GLOBALCONSTANTS IG3_NAME_Functions (* Industry Group 3 specific function defines *)
  (* Standard: 61499-1 *)
  (* Version 1.0, 2026-06-29, Franz Höpfinger, Demmler Andreas Fahrzeugbau *)
  PACKAGE isobus::pgn::const;
  VAR_GLOBAL CONSTANT
    F_SUPPLEMENTAL_ENGINE_CONTROL_SENSING : BYTE := 128; (* Sys: Non-specific system, Func: Supplemental Engine Control Sensing *)
    F_LASER_RECEIVER : BYTE := 129; (* Sys: Non-specific system, Func: Laser Receiver *)
    F_LAND_LEVELING_SYSTEM_OPERATOR_INTERFACE : BYTE := 130; (* Sys: Non-specific system, Func: Land Leveling System Operator Interface - A component that allows *)
    F_LAND_LEVELING_ELECTRIC_MAST : BYTE := 131; (* Sys: Non-specific system, Func: Land Leveling Electric Mast *)
    F_SINGLE_LAND_LEVELING_SYSTEM_SUPERVISOR : BYTE := 132; (* Sys: Non-specific system, Func: Single Land Leveling System Supervisor *)
    F_LAND_LEVELING_SYSTEM_DISPLAY : BYTE := 133; (* Sys: Non-specific system, Func: Land Leveling System Display *)
    F_LASER_TRACER : BYTE := 134; (* Sys: Non-specific system, Func: Laser Tracer *)
    F_LOADER_CONTROL : BYTE := 135; (* Sys: Non-specific system, Func: Loader Control *)
    F_SLOPE_SENSOR : BYTE := 136; (* Sys: Non-specific system, Func: Slope Sensor - Measures the slope along a axis. *)
    F_LIFTARM_CONTROL : BYTE := 137; (* Sys: Non-specific system, Func: Liftarm Control - Controller whose primary purpose is to control *)
    F_SUPPLEMENTAL_SENSOR_PROCESSING_UNITS : BYTE := 138; (* Sys: Non-specific system, Func: Supplemental Sensor Processing Units - An ECU functioning as an *)
    F_HYDRAULIC_SYSTEM_PLANNER : BYTE := 139; (* Sys: Non-specific system, Func: Hydraulic System Planner - Coordinates the functions of a number *)
    F_HYDRAULIC_VALVE_CONTROLLER : BYTE := 140; (* Sys: Non-specific system, Func: Hydraulic Valve Controller - The valve controller will typically *)
    F_JOYSTICK_CONTROL : BYTE := 141; (* Sys: Non-specific system, Func: Joystick Control - Joystick Control *)
    F_ROTATION_SENSOR : BYTE := 142; (* Sys: Non-specific system, Func: Rotation Sensor - A device that measures the rotational angle *)
    F_SONIC_SENSOR : BYTE := 143; (* Sys: Non-specific system, Func: Sonic Sensor - A device that measures distance via ultrasonic *)
    F_SURVEY_TOTAL_STATION_TARGET : BYTE := 144; (* Sys: Non-specific System, Func: Survey Total Station Target - A survey total station target shall *)
    F_HEADING_SENSOR : BYTE := 145; (* Sys: Non-specific System, Func: Heading Sensor - A device that measures vehicle azimuth. *)
    F_ALARM_DEVICE : BYTE := 146; (* Sys: Non-specific System, Func: Alarm device - Device that provides an audible and/or visual *)
    F_NOT_AVAILABLE : BYTE := 255; (* Sys: Non-specific system, Func: Not Available - This assignment can be used until an explicit *)
    F_SKID_STEER_LOADER_MAIN_CONTROLLER : BYTE := 128; (* Sys: Skid Steer Loader, Func: Main Controller *)
    F_SKID_STEER_LOADER_NOT_AVAILABLE : BYTE := 255; (* Sys: Skid Steer Loader, Func: Not Available - This assignment can be used until an explicit *)
    F_ARTICULATED_DUMP_TRUCK_NOT_AVAILABLE : BYTE := 255; (* Sys: Articulated Dump Truck, Func: Not Available - This assignment can be used until an explicit *)
    F_BACKHOE_NOT_AVAILABLE : BYTE := 255; (* Sys: Backhoe, Func: Not Available - This assignment can be used until an explicit function has *)
    F_CRAWLER_BLADE_CONTROLLER : BYTE := 128; (* Sys: Crawler, Func: Blade Controller - Controller for blade height. *)
    F_CRAWLER_NOT_AVAILABLE : BYTE := 255; (* Sys: Crawler, Func: Not Available - This assignment can be used until an explicit function has *)
    F_EXCAVATOR_SLOPE_SENSOR : BYTE := 128; (* Sys: Excavator, Func: Slope Sensor - Measures the slope along a axis. *)
    F_EXCAVATOR_NOT_AVAILABLE : BYTE := 255; (* Sys: Excavator, Func: Not Available - This assignment can be used until an explicit function has *)
    F_FORKLIFT_NOT_AVAILABLE : BYTE := 255; (* Sys: Forklift, Func: Not Available - This assignment can be used until an explicit function has *)
    F_FOUR_WHEEL_DRIVE_LOADER_NOT_AVAILABLE : BYTE := 255; (* Sys: Four Wheel Drive Loader, Func: Not Available - This assignment can be used until an explicit *)
    F_GRADER_HFWD_CONTROLLER : BYTE := 128; (* Sys: Grader, Func: HFWD Controller - Hydraulic front wheel drive controller *)
    F_GRADER_NOT_AVAILABLE : BYTE := 255; (* Sys: Grader, Func: Not Available - This assignment can be used until an explicit function has *)
    F_MILLING_MACHINE_NOT_AVAILABLE : BYTE := 255; (* Sys: Milling Machine, Func: Not Available - The milling machine is used for cutting (or chipping) *)
    F_RECYCLER_AND_SOIL_STABILIZER_NOT_AVAILABLE : BYTE := 255; (* Sys: Recycler and Soil Stabilizer, Func: Not Available - Cold recyclers are used to prepare the *)
    F_BINDING_AGENT_SPREADER_NOT_AVAILABLE : BYTE := 255; (* Sys: Binding Agent Spreader, Func: Not Available - Spreading large quantities of binding agents *)
    F_PAVER_NOT_AVAILABLE : BYTE := 255; (* Sys: Paver, Func: Not Available - A paver (road paver for asphalt or slipform paver for concrete) *)
    F_FEEDER_NOT_AVAILABLE : BYTE := 255; (* Sys: Feeder, Func: Not Available - A feeder is used to convey paver material from a hopper to the *)
    F_SCREENING_PLANT_NOT_AVAILABLE : BYTE := 255; (* Sys: Screening Plant, Func: Not Available - Mobile screening plants are used for screening *)
    F_STACKER_NOT_AVAILABLE : BYTE := 255; (* Sys: Stacker, Func: Not Available - Stackers are used to improve tipping onto conical or *)
    F_ROLLER_NOT_AVAILABLE : BYTE := 255; (* Sys: Roller, Func: Not Available - A roller is used for asphalt and earthwork constuction to *)
    F_CRUSHER_NOT_AVAILABLE : BYTE := 255; (* Sys: Crusher, Func: Not Available - The crusher is used for crushing natural stone and for *)
  END_VAR
END_GLOBALCONSTANTS
